// TIA Portal V20 export
// export: Created 2025-12-01T14:56:15.044482Z, ExportSetting None, DisplayName Totally Integrated Automation Portal, DisplayVersion V20 Update 3, DisplayName TIA Portal Openness, DisplayVersion V20 Update 3, DisplayName TIA Portal Version Control Interface, DisplayVersion V20 Update 3, DisplayName STEP 7 Professional, DisplayVersion V20 Update 3, DisplayName STEP 7 Safety, DisplayVersion V20 Update 2, DisplayName WinCC Basic/Comfort/Advanced, DisplayVersion V20 Update 3, DisplayName WinCC Professional, DisplayVersion V20 Update 3, DisplayName WinCC Unified, DisplayVersion V20 Update 3
TYPE "ROUT_Def_Scanner"
// El 20170522 se incluyen las modificaciones para poder recibir y tratar mensajes INIR para varios bucles.
   STRUCT
      Tipo : UInt := 1;   // Tipo 1 cruce(WS,Cabecera,Sorter) Tipo 2 Validacion Etiqueta en Lista
      Bit_Ini_Ordenes : UInt := 0;   // Bit de Offset para obtener la orden (Tipo 1)
      N_Bits_Orden : UInt := 1;   // Numero de Bits que integran la orden (Max 4 bits)
      Num_Inicializacion : Byte := -1;   // Numero de zona inicialización router asignada
      Libre_Byte : Byte;
      Libre_Word : Byte;
   END_STRUCT;
END_TYPE
